// TIA Portal project "Hiseresis" (V15)

(* hardware
DEVICE "S7-1200 station_1"  S7-1200 Station
   slot 0: "Rack_0"  S7-1200 Rack  Rack  V1.0
   slot 1: "PLC_1"  CPU 1214C DC/DC/DC  6ES7 214-1AG40-0XB0  V4.2
*)

// ===== PLC "PLC_1"  CPU 1214C DC/DC/DC =====

VAR_GLOBAL   // PLC tag table "Tabla de variables estándar"
   "Tag_1" AT 7W64-1 : Int;
   "Tag_2" AT %IW64 : Int;
   "Ventilador" AT %Q0.0 : Bool;
END_VAR

DATA_BLOCK "Mis_datos"   // DB1
{ S7_Optimized_Access := 'TRUE' }
VERSION : 0.1
   VAR
      Temperatura : Real;
      SP : Real;
      SP_Menos : Real;
      SP_Mas : Real;
   END_VAR
BEGIN
END_DATA_BLOCK

FUNCTION "Acondicionamiento" : Void   // FC1, LAD
{ S7_Optimized_Access := 'TRUE' }
VERSION : 0.1
   VAR_TEMP
      Dato1 : Real;
      Dato2 : Real;
   END_VAR
BEGIN

REGION Network 1
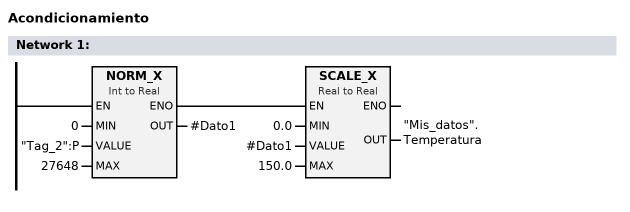
   RUNG wire#powerrail
      { S7_Templates := "[SrcType := Int, DestType := Real]" } Normalize(min := 0, value := "Tag_2":P, max := 27648, out => #Dato1)
      { S7_Templates := "[SrcType := Real, DestType := Real]" } Scale(min := 0.0, value := #Dato1, max := 150.0, out => "Mis_datos".Temperatura)
   END_RUNG
   // the same network as SCL:
   #Dato1 := NORM_X(MIN := 0, VALUE := "Tag_2":P, MAX := 27648);
   "Mis_datos".Temperatura := SCALE_X(MIN := 0.0, VALUE := #Dato1, MAX := 150.0);
END_REGION
END_FUNCTION

FUNCTION "Control_ON_OFF" : Void   // FC2, LAD
{ S7_Optimized_Access := 'TRUE' }
VERSION : 0.1
BEGIN

REGION Network 1
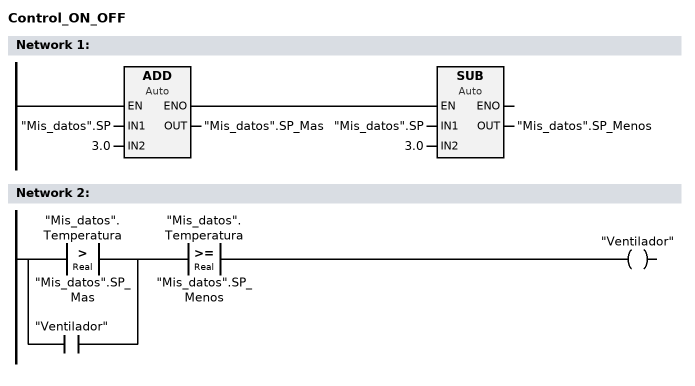
   RUNG wire#powerrail
      Add(in1 := "Mis_datos".SP, in2 := 3.0, out => "Mis_datos".SP_Mas)
      Sub(in1 := "Mis_datos".SP, in2 := 3.0, out => "Mis_datos".SP_Menos)
   END_RUNG
   // the same network as SCL:
   "Mis_datos".SP_Mas := "Mis_datos".SP + 3.0;
   "Mis_datos".SP_Menos := "Mis_datos".SP - 3.0;
END_REGION

REGION Network 2
   RUNG wire#powerrail
      { S7_Templates := "SrcType := Real" } GT_Contact(in1 := "Mis_datos".Temperatura, in2 := "Mis_datos".SP_Mas)
      wire#w1
      { S7_Templates := "SrcType := Real" } GE_Contact(in1 := "Mis_datos".Temperatura, in2 := "Mis_datos".SP_Menos)
      Coil( "Ventilador" )
   END_RUNG
   RUNG wire#powerrail
      Contact( "Ventilador" )
   END_RUNG wire#w1
   // the same network as SCL:
   "Ventilador" := (("Mis_datos".Temperatura > "Mis_datos".SP_Mas) OR "Ventilador") AND ("Mis_datos".Temperatura >= "Mis_datos".SP_Menos);
END_REGION
END_FUNCTION

ORGANIZATION_BLOCK "Main"   // OB1, LAD, ProgramCycle
TITLE = "Main Program Sweep (Cycle)"
{ S7_Optimized_Access := 'TRUE' }
VERSION : 0.1
   VAR_INPUT
      Initial_Call : Bool;   // Initial call of this OB
      Remanence : Bool;   // =True, if remanent data are available
   END_VAR
BEGIN
END_ORGANIZATION_BLOCK